// Block: HMI

DATA_BLOCK HMI
VERSION : 0.1
   NON_RETAIN
   VAR
      PLCDateTime : DTL;
      ProjectInfo : ProjectInfo;
      AreaGen : Struct
         Status : StatusArea;
         Pb_SafetyRstAll : Bool;
         Sgn_SafetyRstAll : Bool;
         Pb_LampTest : Bool;
      END_STRUCT;
   END_VAR

BEGIN
   // No initialization required
END_DATA_BLOCK
